KUKA KRL data list: kappen.dat

&ACCESS RVO
DEFDAT  KAPPEN
SIGNAL PROGRAMM $OUT[57]  TO $OUT[64]
ENDDAT
